{region '#Template'}
	{attribute 'Version' := '1.0.0.0'}
	{attribute 'Tags' := '"LCID": "1031", "Text": "DUT, Operation mode, Universal, Modulation"'}
	{attribute 'Tags' := '"LCID": "1033", "Text": "DUT, Operation mode, Universal, Modulation"'}
	{attribute 'Description' := '"LCID": "1031", "Text": "Modulationsbefehle"'}
	{attribute 'Description' := '"LCID": "1033", "Text": "modulation commands"'}
{endregion}

{attribute 'qualified_only'}
TYPE E_BA_MdltCmd :
(
	eOff			:= 1,
	eOn				:= 2,
	eMin			:= 3,
	eMax			:= 4
	
) UDINT;
END_TYPE

(* stored: Version 1.1.0.1, ProductVersion 3.1.4024.9
   DUT E_BA_MdltCmd: Id {c8bac757-6f17-4014-9aaa-3fcc3890d3b2} *)
